/// EtherCAT IO structure
TYPE ST_EtherCatBoxIO :
STRUCT
	
	/// Data from device.
	aeEtherCatBoxState 		AT %I*	 : E_EtherCatSlaveState;	
	
	/// Data to device.           
	
END_STRUCT
END_TYPE

(* stored: Version 1.1.0.1, ProductVersion 3.1.4022.7
   DUT ST_EtherCatBoxIO: Id {9676ff8a-1d41-4fc4-999b-3917fca72095} *)
